//==================================================================================================
//							Beckhoff Automation Poland
//									25.04.2018
//		Program obslugujacy pamiec nieulotna 
// 	v1.3	|| TC v 3.1.4022.16		|| - Przeniesienie logowania do EvenLogger'a do programu P_SystemDiag_EventLog
// 	v1.2	|| TC v 3.1.4022.0		|| - Dodanie akcji UPS
//	v1.1 	|| TC v 3.1.4020.14 	|| - Dodane wyjscia bOk, bWarning, bError
//	v1.0 	|| TC v 3.1.4020.0 		|| - Pierwsza wersja
//==================================================================================================
PROGRAM P_Persistent
VAR_INPUT
	bWrite						: BOOL;						// Zapis na rozkaz - tylko dla iType = 0 lub nieokreslonego, gdy używany jest FB_WritePersistentData
	tInterval					: TIME := T#1H;				// Czestotliwosc zapisu na karte CF - tylko dla iType = 0 lub nieokreslonego, gdy używany jest FB_WritePersistentData
END_VAR
VAR_OUTPUT
	// Brak obslugi
	bOK							: BOOL := TRUE;				// Brak bledow i ostrzezen
	bWarning					: BOOL;						// Ostrzezenie
	bError						: BOOL;						// Zbiorcza flaga bledow
END_VAR
VAR
	iType						: INT := 0;					(* typ zapisu persistent:
																0: standardowo - na zadanie oraz co okreslony czas
																10: FB_S_UPS, np: CX50x0,C6915-0000,CP62xx-0020,CP77xx-0030
																20: FB_S_UPS_CB3011, np: CP66xx-0020, CP26xx-0000
																30: FB_S_UPS_CX51x0, np: CX51x0
																40: FB_S_UPS_CX9020_U900, np: CX9020 *)
	fbS_UPS						: FB_S_UPS;
	fbS_UPS_CB3011				: FB_S_UPS_CB3011;
	fbS_UPS_CX51x0				: FB_S_UPS_CX51x0;
	fbS_UPS_CX9020_U900			: FB_S_UPS_CX9020_U900;
	fbS_UPS_BAPI				: FB_S_UPS_BAPI;
	// Obsługa ogólna
	fbWritePersistentData 		: FB_WritePersistentData;	// Blok zapisu
	T1							: TON;						// Timer zapisu
END_VAR

CASE iType OF
	0:
		A_WritePersistentData();
		
	10:
	
		A_fbS_UPS();
		
	20:
		
		A_fbS_UPS_CB3011();
		
	30:
	
		A_fbS_UPS_CX51x0();
		
	40:
	
		A_fbS_UPS_CX9020_U900();
		
	50:
	
		A_fbS_UPS_BAPI();
		
ELSE
		A_WritePersistentData();		
		
END_CASE

ACTION A_fbS_UPS:
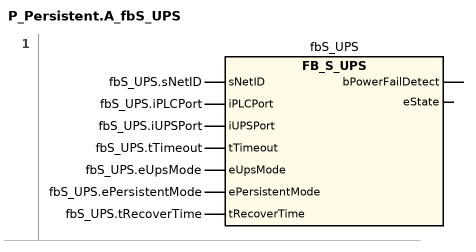
// NETWORK 1
fbS_UPS(
    sNetID := fbS_UPS.sNetID,
    iPLCPort := fbS_UPS.iPLCPort,
    iUPSPort := fbS_UPS.iUPSPort,
    tTimeout := fbS_UPS.tTimeout,
    eUpsMode := fbS_UPS.eUpsMode,
    ePersistentMode := fbS_UPS.ePersistentMode,
    tRecoverTime := fbS_UPS.tRecoverTime); // FB_S_UPS
END_ACTION

ACTION A_fbS_UPS_BAPI:
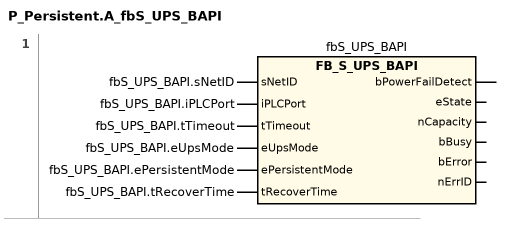
// NETWORK 1
fbS_UPS_BAPI(
    sNetID := fbS_UPS_BAPI.sNetID,
    iPLCPort := fbS_UPS_BAPI.iPLCPort,
    tTimeout := fbS_UPS_BAPI.tTimeout,
    eUpsMode := fbS_UPS_BAPI.eUpsMode,
    ePersistentMode := fbS_UPS_BAPI.ePersistentMode,
    tRecoverTime := fbS_UPS_BAPI.tRecoverTime); // FB_S_UPS_BAPI
END_ACTION

ACTION A_fbS_UPS_CB3011:
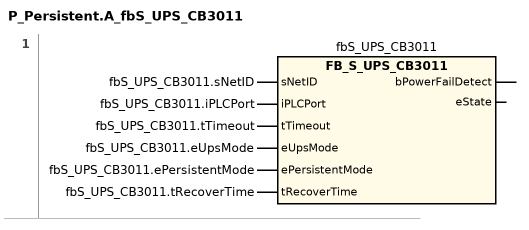
// NETWORK 1
fbS_UPS_CB3011(
    sNetID := fbS_UPS_CB3011.sNetID,
    iPLCPort := fbS_UPS_CB3011.iPLCPort,
    tTimeout := fbS_UPS_CB3011.tTimeout,
    eUpsMode := fbS_UPS_CB3011.eUpsMode,
    ePersistentMode := fbS_UPS_CB3011.ePersistentMode,
    tRecoverTime := fbS_UPS_CB3011.tRecoverTime); // FB_S_UPS_CB3011
END_ACTION

ACTION A_fbS_UPS_CX51x0:
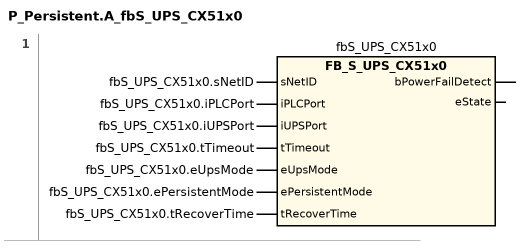
// NETWORK 1
fbS_UPS_CX51x0(
    sNetID := fbS_UPS_CX51x0.sNetID,
    iPLCPort := fbS_UPS_CX51x0.iPLCPort,
    iUPSPort := fbS_UPS_CX51x0.iUPSPort,
    tTimeout := fbS_UPS_CX51x0.tTimeout,
    eUpsMode := fbS_UPS_CX51x0.eUpsMode,
    ePersistentMode := fbS_UPS_CX51x0.ePersistentMode,
    tRecoverTime := fbS_UPS_CX51x0.tRecoverTime); // FB_S_UPS_CX51x0
END_ACTION

ACTION A_fbS_UPS_CX9020_U900:
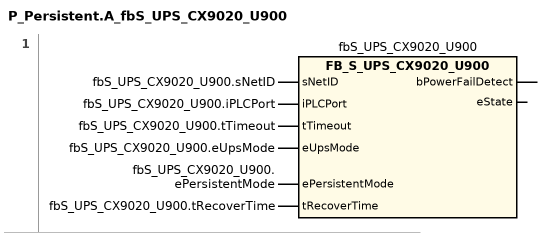
// NETWORK 1
fbS_UPS_CX9020_U900(
    sNetID := fbS_UPS_CX9020_U900.sNetID,
    iPLCPort := fbS_UPS_CX9020_U900.iPLCPort,
    tTimeout := fbS_UPS_CX9020_U900.tTimeout,
    eUpsMode := fbS_UPS_CX9020_U900.eUpsMode,
    ePersistentMode := fbS_UPS_CX9020_U900.ePersistentMode,
    tRecoverTime := fbS_UPS_CX9020_U900.tRecoverTime); // FB_S_UPS_CX9020_U900
END_ACTION

ACTION A_WritePersistentData:
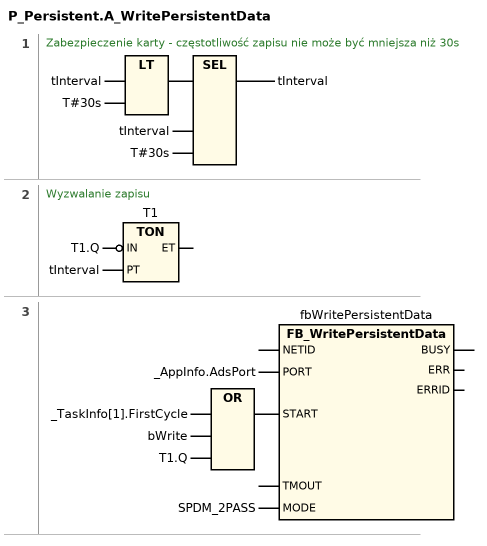
// NETWORK 1
// Zabezpieczenie karty - częstotliwość zapisu nie może być mniejsza niż 30s
tInterval := SEL(tInterval < T#30s, tInterval, T#30s);

// NETWORK 2
// Wyzwalanie zapisu
T1(IN := NOT T1.Q, PT := tInterval); // TON

// NETWORK 3
fbWritePersistentData(
    PORT := _AppInfo.AdsPort,
    START := _TaskInfo[1].FirstCycle OR bWrite OR T1.Q,
    MODE := SPDM_2PASS); // FB_WritePersistentData
END_ACTION

END_PROGRAM

(* stored: Version 1.1.0.1, ProductVersion 3.1.4022.12
   POU P_Persistent: Id {188d73a3-0452-479f-b48c-0ee7551b4de1}, SpecialFunc None
   Action A_fbS_UPS: Id {8b222a48-c306-4706-9d37-e32da7b93a34}
   Action A_fbS_UPS_BAPI: Id {af48fac2-ce8b-4607-8e0a-49a7299bcf3a}
   Action A_fbS_UPS_CB3011: Id {4240ce2d-4cb7-49af-8c56-ac9a76010f70}
   Action A_fbS_UPS_CX51x0: Id {88db6106-cabd-4b4c-b4f8-cd49e3cad3b2}
   Action A_fbS_UPS_CX9020_U900: Id {b44081b3-05fd-45ca-8206-461be1a03847}
   Action A_WritePersistentData: Id {f1d20de6-e870-4621-8c24-2223b1c9304b} *)
